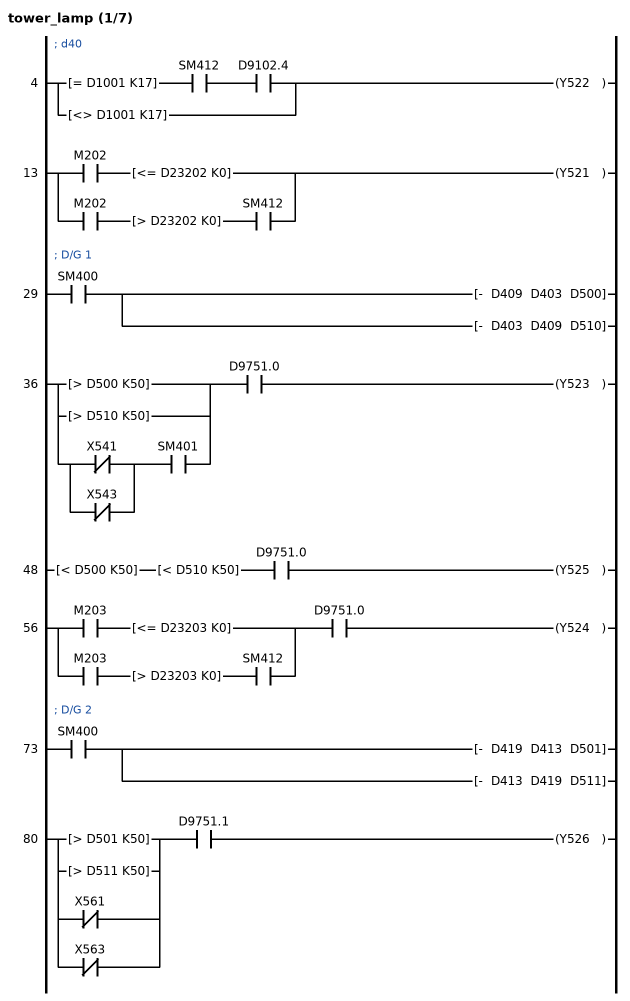
[picture p312: ladder of tower_lamp, rungs at steps 4 to 80]
; d40
4     LD=     D1001 K17
      AND     SM412
      AND     D9102.4
      OR<>    D1001 K17
      OUT     Y522
13    LD      M202
      AND<=   D23202 K0
      LD      M202
      AND>    D23202 K0
      AND     SM412
      ORB
      OUT     Y521
; D/G 1
29    LD      SM400
      -       D409 D403 D500
      -       D403 D409 D510
36    LD>     D500 K50
      OR>     D510 K50
      LDI     X541
      ORI     X543
      AND     SM401
      ORB
      AND     D9751.0
      OUT     Y523
48    LD<     D500 K50
      AND<    D510 K50
      AND     D9751.0
      OUT     Y525
56    LD      M203
      AND<=   D23203 K0
      LD      M203
      AND>    D23203 K0
      AND     SM412
      ORB
      AND     D9751.0
      OUT     Y524
; D/G 2
73    LD      SM400
      -       D419 D413 D501
      -       D413 D419 D511
80    LD>     D501 K50
      OR>     D511 K50
      ORI     X561
      ORI     X563
      AND     D9751.1
      OUT     Y526
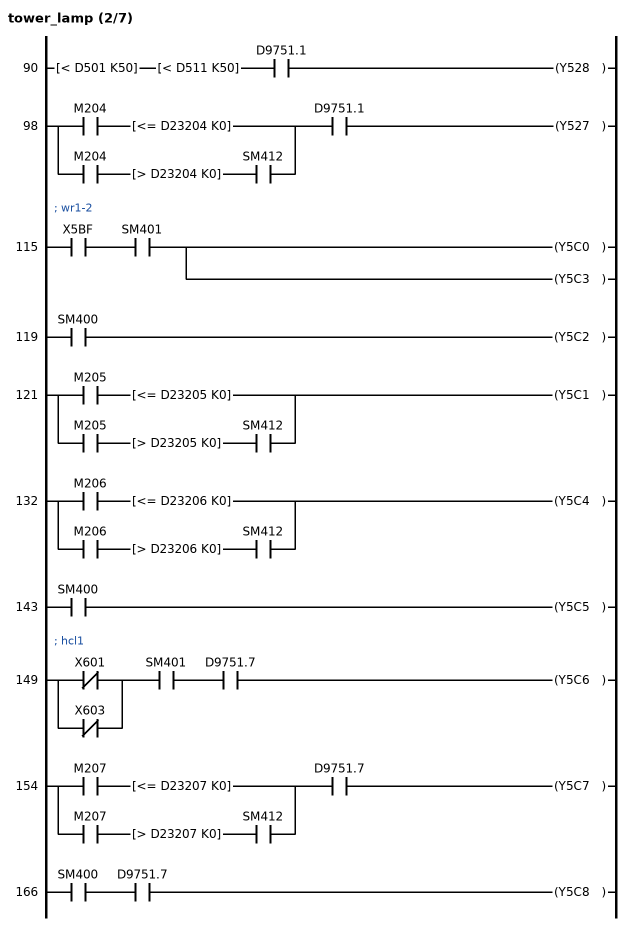
90    LD<     D501 K50
      AND<    D511 K50
      AND     D9751.1
      OUT     Y528
98    LD      M204
      AND<=   D23204 K0
      LD      M204
      AND>    D23204 K0
      AND     SM412
      ORB
      AND     D9751.1
      OUT     Y527
; wr1-2
115   LD      X5BF
      AND     SM401
      OUT     Y5C0
      OUT     Y5C3
119   LD      SM400
      OUT     Y5C2
121   LD      M205
      AND<=   D23205 K0
      LD      M205
      AND>    D23205 K0
      AND     SM412
      ORB
      OUT     Y5C1
132   LD      M206
      AND<=   D23206 K0
      LD      M206
      AND>    D23206 K0
      AND     SM412
      ORB
      OUT     Y5C4
143   LD      SM400
      OUT     Y5C5
; hcl1
149   LDI     X601
      ORI     X603
      AND     SM401
      AND     D9751.7
      OUT     Y5C6
154   LD      M207
      AND<=   D23207 K0
      LD      M207
      AND>    D23207 K0
      AND     SM412
      ORB
      AND     D9751.7
      OUT     Y5C7
166   LD      SM400
      AND     D9751.7
      OUT     Y5C8
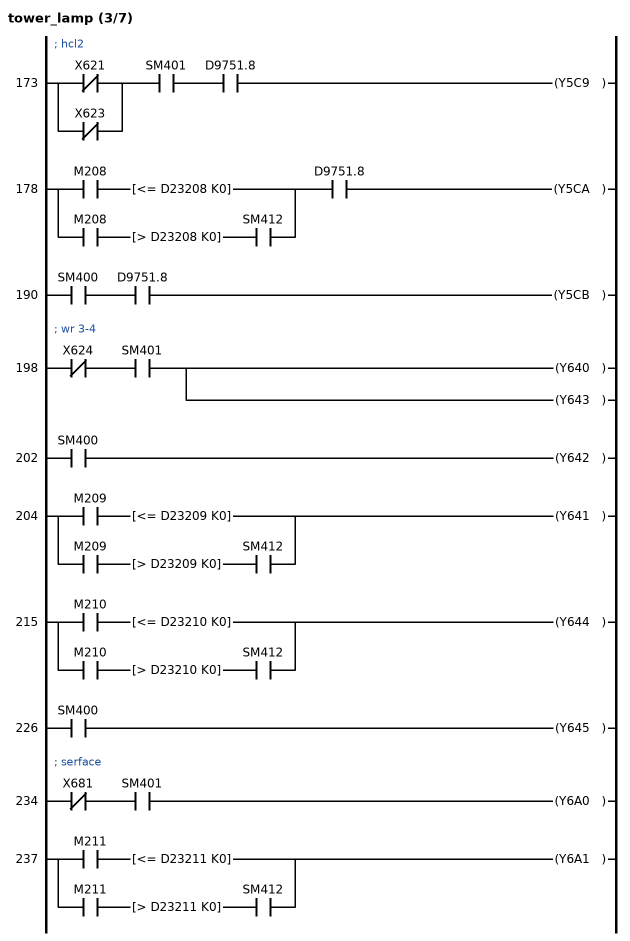
; hcl2
173   LDI     X621
      ORI     X623
      AND     SM401
      AND     D9751.8
      OUT     Y5C9
178   LD      M208
      AND<=   D23208 K0
      LD      M208
      AND>    D23208 K0
      AND     SM412
      ORB
      AND     D9751.8
      OUT     Y5CA
190   LD      SM400
      AND     D9751.8
      OUT     Y5CB
; wr 3-4
198   LDI     X624
      AND     SM401
      OUT     Y640
      OUT     Y643
202   LD      SM400
      OUT     Y642
204   LD      M209
      AND<=   D23209 K0
      LD      M209
      AND>    D23209 K0
      AND     SM412
      ORB
      OUT     Y641
215   LD      M210
      AND<=   D23210 K0
      LD      M210
      AND>    D23210 K0
      AND     SM412
      ORB
      OUT     Y644
226   LD      SM400
      OUT     Y645
; serface
234   LDI     X681
      AND     SM401
      OUT     Y6A0
237   LD      M211
      AND<=   D23211 K0
      LD      M211
      AND>    D23211 K0
      AND     SM412
      ORB
      OUT     Y6A1
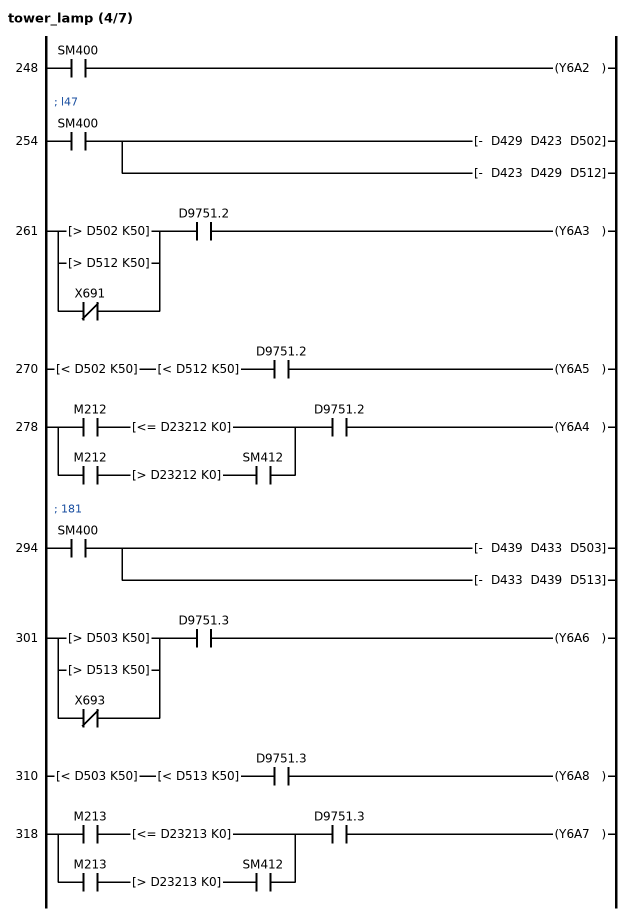
248   LD      SM400
      OUT     Y6A2
; l47
254   LD      SM400
      -       D429 D423 D502
      -       D423 D429 D512
261   LD>     D502 K50
      OR>     D512 K50
      ORI     X691
      AND     D9751.2
      OUT     Y6A3
270   LD<     D502 K50
      AND<    D512 K50
      AND     D9751.2
      OUT     Y6A5
278   LD      M212
      AND<=   D23212 K0
      LD      M212
      AND>    D23212 K0
      AND     SM412
      ORB
      AND     D9751.2
      OUT     Y6A4
; 181
294   LD      SM400
      -       D439 D433 D503
      -       D433 D439 D513
301   LD>     D503 K50
      OR>     D513 K50
      ORI     X693
      AND     D9751.3
      OUT     Y6A6
310   LD<     D503 K50
      AND<    D513 K50
      AND     D9751.3
      OUT     Y6A8
318   LD      M213
      AND<=   D23213 K0
      LD      M213
      AND>    D23213 K0
      AND     SM412
      ORB
      AND     D9751.3
      OUT     Y6A7
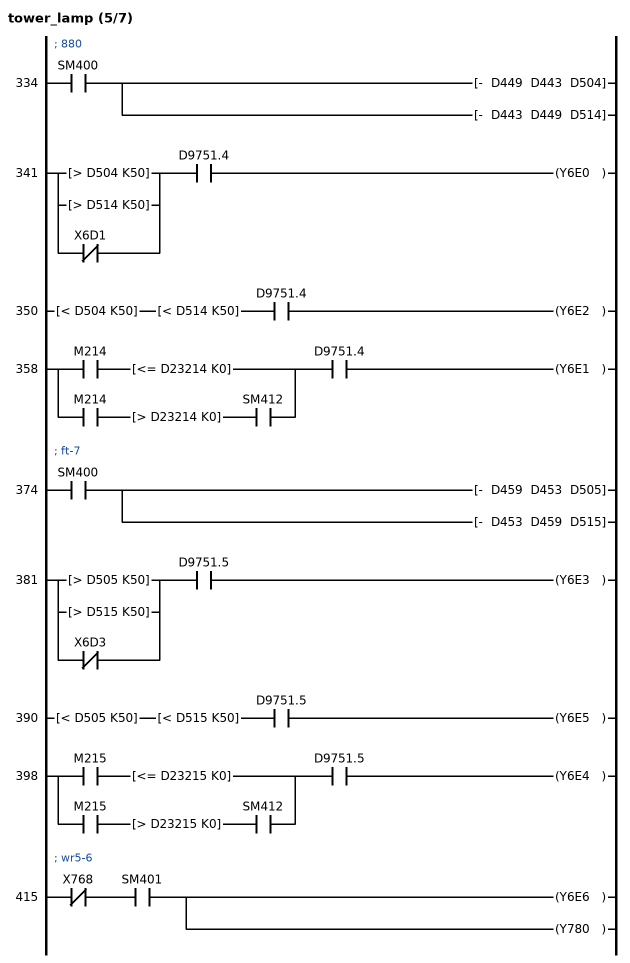
; 880
334   LD      SM400
      -       D449 D443 D504
      -       D443 D449 D514
341   LD>     D504 K50
      OR>     D514 K50
      ORI     X6D1
      AND     D9751.4
      OUT     Y6E0
350   LD<     D504 K50
      AND<    D514 K50
      AND     D9751.4
      OUT     Y6E2
358   LD      M214
      AND<=   D23214 K0
      LD      M214
      AND>    D23214 K0
      AND     SM412
      ORB
      AND     D9751.4
      OUT     Y6E1
; ft-7
374   LD      SM400
      -       D459 D453 D505
      -       D453 D459 D515
381   LD>     D505 K50
      OR>     D515 K50
      ORI     X6D3
      AND     D9751.5
      OUT     Y6E3
390   LD<     D505 K50
      AND<    D515 K50
      AND     D9751.5
      OUT     Y6E5
398   LD      M215
      AND<=   D23215 K0
      LD      M215
      AND>    D23215 K0
      AND     SM412
      ORB
      AND     D9751.5
      OUT     Y6E4
; wr5-6
415   LDI     X768
      AND     SM401
      OUT     Y6E6
      OUT     Y780
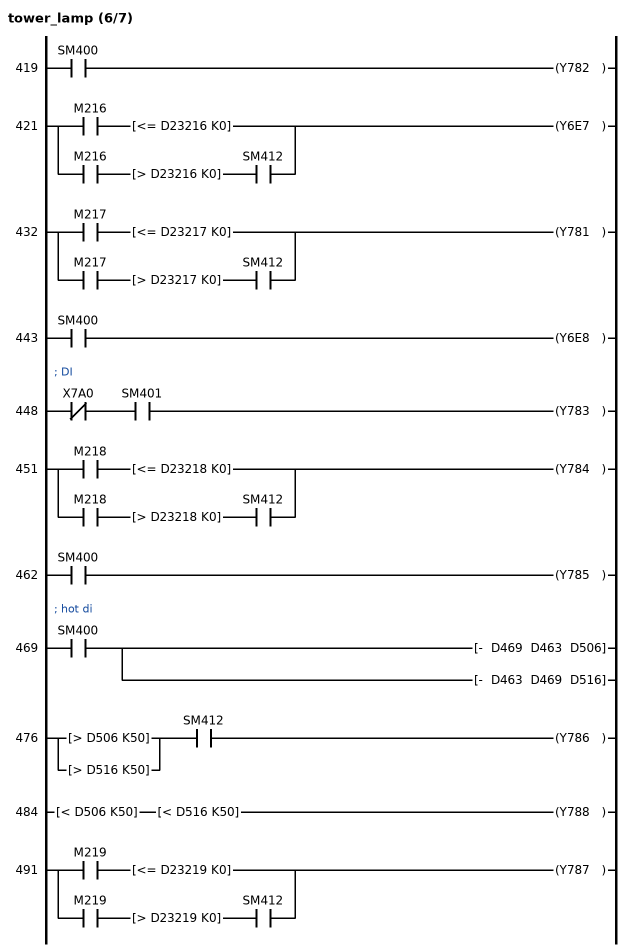
419   LD      SM400
      OUT     Y782
421   LD      M216
      AND<=   D23216 K0
      LD      M216
      AND>    D23216 K0
      AND     SM412
      ORB
      OUT     Y6E7
432   LD      M217
      AND<=   D23217 K0
      LD      M217
      AND>    D23217 K0
      AND     SM412
      ORB
      OUT     Y781
443   LD      SM400
      OUT     Y6E8
; DI
448   LDI     X7A0
      AND     SM401
      OUT     Y783
451   LD      M218
      AND<=   D23218 K0
      LD      M218
      AND>    D23218 K0
      AND     SM412
      ORB
      OUT     Y784
462   LD      SM400
      OUT     Y785
; hot di
469   LD      SM400
      -       D469 D463 D506
      -       D463 D469 D516
476   LD>     D506 K50
      OR>     D516 K50
      AND     SM412
      OUT     Y786
484   LD<     D506 K50
      AND<    D516 K50
      OUT     Y788
491   LD      M219
      AND<=   D23219 K0
      LD      M219
      AND>    D23219 K0
      AND     SM412
      ORB
      OUT     Y787
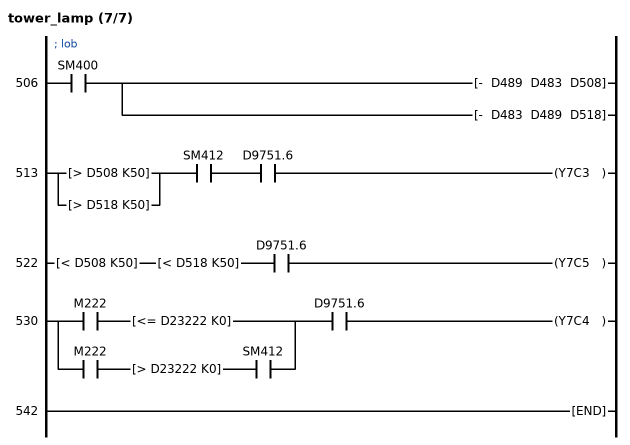
; lob
506   LD      SM400
      -       D489 D483 D508
      -       D483 D489 D518
513   LD>     D508 K50
      OR>     D518 K50
      AND     SM412
      AND     D9751.6
      OUT     Y7C3
522   LD<     D508 K50
      AND<    D518 K50
      AND     D9751.6
      OUT     Y7C5
530   LD      M222
      AND<=   D23222 K0
      LD      M222
      AND>    D23222 K0
      AND     SM412
      ORB
      AND     D9751.6
      OUT     Y7C4
542   END
END_PROGRAM

PROGRAM unload
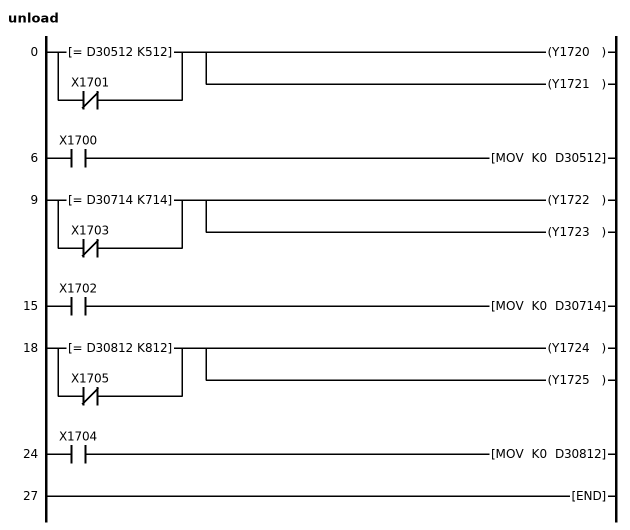
0     LD=     D30512 K512
      ORI     X1701
      OUT     Y1720
      OUT     Y1721
6     LD      X1700
      MOV     K0 D30512
9     LD=     D30714 K714
      ORI     X1703
      OUT     Y1722
      OUT     Y1723
15    LD      X1702
      MOV     K0 D30714
18    LD=     D30812 K812
      ORI     X1705
      OUT     Y1724
      OUT     Y1725
24    LD      X1704
      MOV     K0 D30812
27    END
END_PROGRAM

PROGRAM water_supply
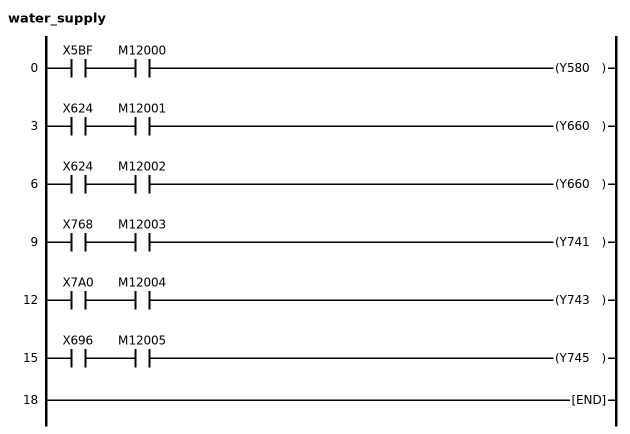
0     LD      X5BF
      AND     M12000
      OUT     Y580
3     LD      X624
      AND     M12001
      OUT     Y660
6     LD      X624
      AND     M12002
      OUT     Y660
9     LD      X768
      AND     M12003
      OUT     Y741
12    LD      X7A0
      AND     M12004
      OUT     Y743
15    LD      X696
      AND     M12005
      OUT     Y745
18    END
END_PROGRAM

// device comments not shown above
X2B0  ; cover D40 open
X2B1  ; cover D40 close
X2B2  ; cover D40 hi
X2B3  ; cover D40 low
B2B0  ; cover D40 open
B2B1  ; cover D40 close
B2B2  ; cover D40 hi
B2B3  ; cover D40 low
